TYPE ST_InterlockList :
STRUCT
	arr_Interlocks : ARRAY[0..GVL.g_nLEN_INTERLOCK_LIST-1] OF ST_Interlock;
END_STRUCT
END_TYPE

(* stored: Version 1.1.0.1, ProductVersion 3.1.4024.12
   DUT ST_InterlockList: Id {7ab115a9-8ad9-4d57-b427-1634f5f82e75} *)
